ABB RobotStudio station: Task1.rspag

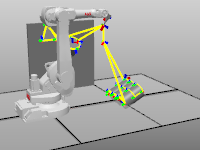
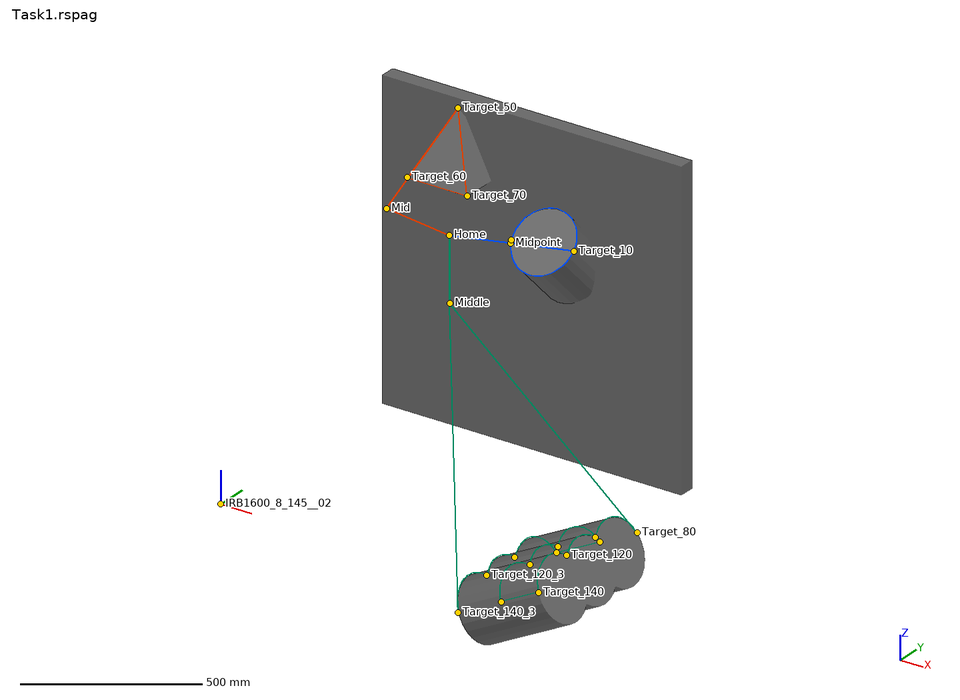
[picture v1: parts stored in the station drawn from their meshes, with robot base, taught points and paths (robot models come from the ABB library and are not in the file)]
--- station ---
Station Task1 (saved by RobotStudio 21.4.9700.0)
Controller IRB1600_8_145
  mechanical unit ROB_1: IRB1600_8_145__02, 6 joints, base frame (0, 0, 0) mm
Layout (positions relative to the parent item):
  - IRB1600_8_145__02 [mechanism, from Robots\IRB1600_8_145_G_02.rslib] at (0, 0, 0) mm; joint values [0, 0, 0, 0, 0.5236, 0] (rad or m)
  - MyNewTool [mechanism] at (806.29, 0, 1154) mm, rotated rx 180 ry 60 rz 180 deg
      TCP MyNewTool at (127, 0, 25) mm
      links: Part_1
  - Wall [part] at (0, 770.01, 0) mm, size 1000 x 50 x 1000 mm
  - Cylinder [part] at (612.14, 809.48, 561.49) mm, rotated rx 45.02 ry 0 rz 0 deg, size 200 x 199.7 x 200 mm
  - Pyramid [part] at (264.87, 755.65, 778.7) mm, size 200 x 200 x 200 mm
  - Roll [part] at (970.39, 135.85, 7.21) mm, rotated rx 0 ry -7.05 rz 0 deg, size 350.3 x 473.3 x 290.5 mm
Attachment: MyNewTool is attached to IRB1600_8_145__02 / Link6
Attachment: Pyramid is attached to Wall
Attachment: Cylinder is attached to Wall
Attachment: Workobject_Cylinder is attached to Cylinder
Attachment: Workobject_Pyramid is attached to Pyramid
Attachment: Workobject_Roll is attached to Roll
Collision set CollisionSet_1: MyNewTool against Wall, Pyramid, Cylinder, Roll, near miss 0 m

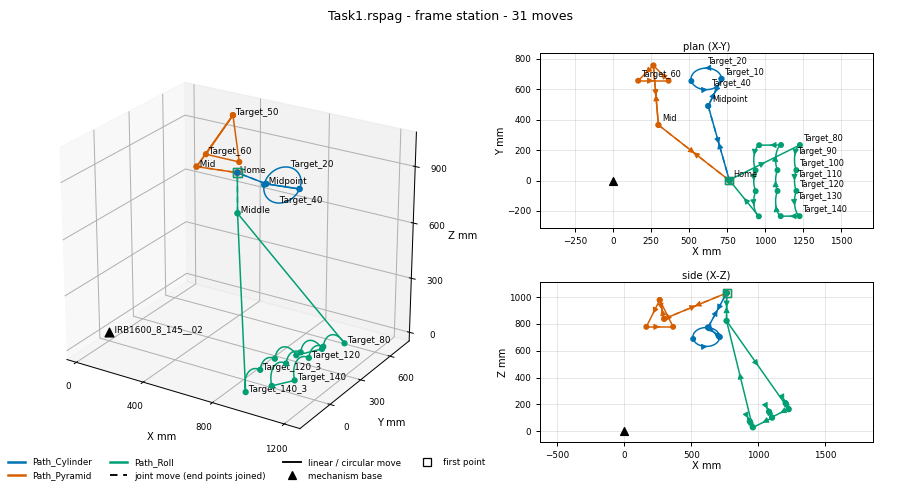
[picture p0: tool path of Task1.rspag in frame station, 31 of 31 moves have a stored position in this frame; points joined in program order, loops and branches not executed]
--- Backups/IRB1600_8_145/RAPID/TASK1/PROGMOD/CalibData.mod ---
MODULE CalibData
    PERS tooldata MyNewTool:=[TRUE,[[127,0,25],[1,0,0,0]],[1,[0,0,1],[1,0,0,0],0,0,0]];
    TASK PERS wobjdata Workobject_Cylinder:=[FALSE,TRUE,"",[[612.143,668.01,702.868],[1,0,0,0]],[[0,0,0],[1,0,0,0]]];
    TASK PERS wobjdata Workobject_Pyramid:=[FALSE,TRUE,"",[[264.868,755.646,978.698540948],[1,0,0,0]],[[0,0,0],[1,0,0,0]]];
    TASK PERS wobjdata Workobject_Roll:=[FALSE,TRUE,"",[[1192.676351946,151.722,231.573663643],[0.998108504,0,-0.061476934,0]],[[0,0,0],[1,0,0,0]]];
ENDMODULE

--- Backups/IRB1600_8_145/RAPID/TASK1/PROGMOD/Module1.mod ---
MODULE Module1
        CONST robtarget Home:=[[764.442286341,0,1031.514773719],[0.5,0,0.866025404,0],[0,0,0,0],[9E+09,9E+09,9E+09,9E+09,9E+09,9E+09]];
    CONST robtarget Midpoint:=[[12.973976789,-178.364696048,70.89735062],[0.499999992,0.000000012,0.866025408,0.000000063],[0,-1,1,0],[9E+09,9E+09,9E+09,9E+09,9E+09,9E+09]];
    CONST robtarget Target_10:=[[100.000029686,0.000444541,0.000129619],[0.203332137,0.677241495,0.677241495,-0.203332137],[0,-1,1,0],[9E+09,9E+09,9E+09,9E+09,9E+09,9E+09]];
    CONST robtarget Target_20:=[[-10.452816641,70.300573395,70.346628371],[0.203332137,0.677241495,0.677241495,-0.203332137],[0,-1,1,0],[9E+09,9E+09,9E+09,9E+09,9E+09,9E+09]];
    CONST robtarget Target_30:=[[-97.814730387,-14.696284333,-14.706293202],[0.203332137,0.677241495,0.677241495,-0.203332137],[0,-1,1,0],[9E+09,9E+09,9E+09,9E+09,9E+09,9E+09]];
    CONST robtarget Target_40:=[[10.452876013,-70.299684314,-70.346369133],[0.203332137,0.677241495,0.677241495,-0.203332137],[0,-1,1,0],[9E+09,9E+09,9E+09,9E+09,9E+09,9E+09]];
    CONST robtarget Mid:=[[32.899890848,-390.522224232,-140.517124947],[0.500000029,0.000000028,0.866025387,0.000000005],[0,-1,0,0],[9E+09,9E+09,9E+09,9E+09,9E+09,9E+09]];
    CONST robtarget Target_50:=[[0.000271397,-0.000070668,0.000243746],[0.677313487,-0.170224297,0.178019,0.693238318],[0,-3,2,0],[9E+09,9E+09,9E+09,9E+09,9E+09,9E+09]];
    CONST robtarget Target_60:=[[-99.999476706,-99.999818771,-199.999756254],[0.677313487,-0.170224297,0.178019,0.693238318],[0,-3,2,0],[9E+09,9E+09,9E+09,9E+09,9E+09,9E+09]];
    CONST robtarget Target_70:=[[100.000019499,-99.999818771,-199.999756254],[0.677313487,-0.170224297,0.178019,0.693238318],[0,-3,2,0],[9E+09,9E+09,9E+09,9E+09,9E+09,9E+09]];
    CONST robtarget Middle:=[[-353.263741952,-148.821758196,640.167392316],[0.500000003,-0.000000145,0.866025402,-0.000000005],[0,-1,0,0],[9E+09,9E+09,9E+09,9E+09,9E+09,9E+09]];
    CONST robtarget Target_80:=[[26.326445515,81.731014415,-72.332275036],[0.332856556,-0.701020572,0.622776813,0.099627863],[0,0,-2,0],[9E+09,9E+09,9E+09,9E+09,9E+09,9E+09]];
    CONST robtarget Target_90:=[[-0.129173031,-2.554828649,0.353939502],[0.571752943,-0.563857345,0.415379699,0.427344325],[0,1,-2,0],[9E+09,9E+09,9E+09,9E+09,9E+09,9E+09]];
    CONST robtarget Target_100:=[[8.693425716,-83.713774231,-23.885951324],[0.571752943,-0.563857345,0.415379699,0.427344325],[-1,0,-2,0],[9E+09,9E+09,9E+09,9E+09,9E+09,9E+09]];
    CONST robtarget Target_110:=[[-0.430078891,-153.21028872,1.180671556],[0.571752943,-0.563857345,0.415379699,0.427344325],[-1,0,-2,0],[9E+09,9E+09,9E+09,9E+09,9E+09,9E+09]];
    CONST robtarget Target_120:=[[9.059267937,-220.378372878,-24.891094565],[0.571752943,-0.563857345,0.415379699,0.427344325],[-1,0,-2,0],[9E+09,9E+09,9E+09,9E+09,9E+09,9E+09]];
    CONST robtarget Target_130:=[[-0.370119552,-295.624451185,1.015934626],[0.571752943,-0.563857345,0.415379699,0.427344325],[-1,0,-2,0],[9E+09,9E+09,9E+09,9E+09,9E+09,9E+09]];
    CONST robtarget Target_140:=[[24.682445849,-385.928812513,-67.815423077],[0.613657304,-0.513869184,0.350523087,0.486309306],[-1,0,-2,0],[9E+09,9E+09,9E+09,9E+09,9E+09,9E+09]];
    CONST robtarget Target_140_2:=[[-106.175768675,-385.93224335,-115.263854081],[0.61677152,-0.50949384,0.345013933,0.490891338],[-1,0,-2,0],[9E+09,9E+09,9E+09,9E+09,9E+09,9E+09]];
    CONST robtarget Target_130_2:=[[-131.228334076,-295.627882022,-46.432496378],[0.571752943,-0.563857345,0.415379699,0.427344325],[-1,0,-2,0],[9E+09,9E+09,9E+09,9E+09,9E+09,9E+09]];
    CONST robtarget Target_120_2:=[[-121.798946587,-220.381803715,-72.339525569],[0.571752943,-0.563857345,0.415379699,0.427344325],[-1,0,-2,0],[9E+09,9E+09,9E+09,9E+09,9E+09,9E+09]];
    CONST robtarget Target_110_2:=[[-131.288293415,-153.213719557,-46.267759448],[0.571752943,-0.563857345,0.415379699,0.427344325],[-1,0,-2,0],[9E+09,9E+09,9E+09,9E+09,9E+09,9E+09]];
    CONST robtarget Target_100_2:=[[-122.164788808,-83.717205068,-71.334382328],[0.571752943,-0.563857345,0.415379699,0.427344325],[-1,0,-2,0],[9E+09,9E+09,9E+09,9E+09,9E+09,9E+09]];
    CONST robtarget Target_90_2:=[[-130.987387555,-2.558259486,-47.094491502],[0.571752943,-0.563857345,0.415379699,0.427344325],[0,1,-2,0],[9E+09,9E+09,9E+09,9E+09,9E+09,9E+09]];
    CONST robtarget Target_80_2:=[[-104.531769009,81.727583578,-119.78070604],[0.332856556,-0.701020572,0.622776813,0.099627863],[0,1,-3,0],[9E+09,9E+09,9E+09,9E+09,9E+09,9E+09]];
    CONST robtarget Target_80_3:=[[-255.902672948,80.401776355,-173.854840306],[0.332856556,-0.701020572,0.622776813,0.099627863],[0,1,-3,0],[9E+09,9E+09,9E+09,9E+09,9E+09,9E+09]];
    CONST robtarget Target_90_3:=[[-282.358291494,-3.884066709,-101.168625768],[0.571752943,-0.563857345,0.415379699,0.427344325],[0,1,-3,0],[9E+09,9E+09,9E+09,9E+09,9E+09,9E+09]];
    CONST robtarget Target_100_3:=[[-273.535692747,-85.043012291,-125.408516594],[0.571752943,-0.563857345,0.415379699,0.427344325],[-1,0,-3,0],[9E+09,9E+09,9E+09,9E+09,9E+09,9E+09]];
    CONST robtarget Target_110_3:=[[-282.659197354,-154.53952678,-100.341893714],[0.571752943,-0.563857345,0.415379699,0.427344325],[-1,0,-3,0],[9E+09,9E+09,9E+09,9E+09,9E+09,9E+09]];
    CONST robtarget Target_120_3:=[[-273.169850526,-221.707610938,-126.413659835],[0.571752943,-0.563857345,0.415379699,0.427344325],[-1,0,-3,0],[9E+09,9E+09,9E+09,9E+09,9E+09,9E+09]];
    CONST robtarget Target_130_3:=[[-282.599238015,-296.953689245,-100.506630644],[0.571752943,-0.563857345,0.415379699,0.427344325],[-1,0,-3,0],[9E+09,9E+09,9E+09,9E+09,9E+09,9E+09]];
    CONST robtarget Target_140_3:=[[-257.546672614,-387.258050573,-169.337988347],[0.61677152,-0.50949384,0.345013933,0.490891338],[-1,0,-3,0],[9E+09,9E+09,9E+09,9E+09,9E+09,9E+09]];
!***********************************************************
    !
    ! Module:  Module1
    !
    ! Description:
    !   <Insert description here>
    !
    ! Author: ramni
    !
    ! Version: 1.0
    !
    !***********************************************************


    !***********************************************************
    !
    ! Procedure main
    !
    !   This is the entry point of your program
    !
    !***********************************************************
    PROC main()
        !Add your code here
    ENDPROC
    PROC Path_Cylinder()
        MoveJ Home,v1000,fine,MyNewTool\WObj:=wobj0;
        MoveL Midpoint,v1000,fine,MyNewTool\WObj:=Workobject_Cylinder;
        MoveL Target_10,v1000,z10,MyNewTool\WObj:=Workobject_Cylinder;
        MoveC Target_20,Target_30,v100,z10,MyNewTool\WObj:=Workobject_Cylinder;
        MoveC Target_40,Target_10,v100,z10,MyNewTool\WObj:=Workobject_Cylinder;
        MoveL Midpoint,v1000,fine,MyNewTool\WObj:=Workobject_Cylinder;
        MoveJ Home,v1000,fine,MyNewTool\WObj:=wobj0;
        Path_Pyramid;
    ENDPROC
    PROC Path_Pyramid()
        MoveJ Home,v1000,fine,MyNewTool\WObj:=wobj0;
        MoveL Mid,v1000,fine,MyNewTool\WObj:=Workobject_Pyramid;
        MoveL Target_50,v100,z10,MyNewTool\WObj:=Workobject_Pyramid;
        MoveL Target_60,v100,z10,MyNewTool\WObj:=Workobject_Pyramid;
        MoveL Target_70,v100,z10,MyNewTool\WObj:=Workobject_Pyramid;
        MoveL Target_50,v100,z10,MyNewTool\WObj:=Workobject_Pyramid;
        MoveL Mid,v1000,fine,MyNewTool\WObj:=Workobject_Pyramid;
        MoveJ Home,v1000,fine,MyNewTool\WObj:=wobj0;
        Path_Roll;
    ENDPROC
    PROC Path_Roll()
        MoveJ Home,v1000,fine,MyNewTool\WObj:=wobj0;
        MoveL Middle,v1000,fine,MyNewTool\WObj:=Workobject_Roll;
        MoveL Target_80,v100,z10,MyNewTool\WObj:=Workobject_Roll;
        MoveC Target_90,Target_100,v100,z10,MyNewTool\WObj:=Workobject_Roll;
        MoveC Target_110,Target_120,v100,z10,MyNewTool\WObj:=Workobject_Roll;
        MoveC Target_130,Target_140,v100,z10,MyNewTool\WObj:=Workobject_Roll;
        MoveL Target_140_2,v100,z10,MyNewTool\WObj:=Workobject_Roll;
        MoveC Target_130_2,Target_120_2,v100,z10,MyNewTool\WObj:=Workobject_Roll;
        MoveC Target_110_2,Target_100_2,v100,z10,MyNewTool\WObj:=Workobject_Roll;
        MoveC Target_90_2,Target_80_2,v100,z10,MyNewTool\WObj:=Workobject_Roll;
        MoveL Target_80_3,v100,z10,MyNewTool\WObj:=Workobject_Roll;
        MoveC Target_90_3,Target_100_3,v100,z10,MyNewTool\WObj:=Workobject_Roll;
        MoveC Target_110_3,Target_120_3,v100,z10,MyNewTool\WObj:=Workobject_Roll;
        MoveC Target_130_3,Target_140_3,v100,z10,MyNewTool\WObj:=Workobject_Roll;
        MoveL Middle,v1000,fine,MyNewTool\WObj:=Workobject_Roll;
        MoveJ Home,v1000,fine,MyNewTool\WObj:=wobj0;
    ENDPROC
ENDMODULE
